// TIA Portal V20 export
DATA_BLOCK "HmiInterface"   // DB99
// stored: Access Published, MemoryReserve 100, Namespace Unit1.Em10
   VAR
      em : "LAF_typeEmInterface";
      laserMark : "LER_typeSequenceInterface";
      cmLaserMarkJRDetect : "LBC_typeDigitalSignalInterface";
      cmLaserMarkStageLiftUpDown : "LBC_typeTwoWayActuatorInterface";
      cmLaserMarkCoverUpDown : "LBC_typeTwoWayActuatorInterface";
      cmLaserMarkControl : "LER_typeLaserMarkInterface";
      cmQrFixReaderControl : "LER_typeSRX300Interface";
   END_VAR
   VAR RETAIN
      cmLaserMarkHistory : "LER_typeLaserMarkHistory";
   END_VAR
   VAR
      intCondition : "Unit1.Em10.typeIntConditionHmiInterface";
   END_VAR
BEGIN
END_DATA_BLOCK
